Fanuc KAREL source: kt00498.KL

-- PROVISIONAL review KL for V770-1; original PC SHA256 b7b7ee6dab29da864770a4dc023898f2a03b7aa2bf29e70d1882a8a437d3fbb2
-- Incomplete behavior may be omitted. Consult companion uncertainty JSON. Do not deploy.
PROGRAM KT00498
%NOLOCKGROUP
VAR
  OUT : BOOLEAN
-- UNRESOLVED_DECL P1 type=000102
-- UNRESOLVED_DECL P2 type=000102
BEGIN
  -- UNRESOLVED_PC offsets 5-20; opcodes 2E,22,32,35
  -- UNRESOLVED_PC offsets 25-40; opcodes 2E,22,32,35
  -- UNRESOLVED_PC offsets 45-60; opcodes 2E,22,32,35
  -- UNRESOLVED_PC offsets 65-80; opcodes 2E,22,32,35
  -- UNRESOLVED_PC offsets 85-118; opcodes 49,7E,49,7E,AC,23
  -- UNRESOLVED_PC offsets 123-127; opcodes 7F
END KT00498
